// TwinCAT 3 PLC project ControlExtrusora
// ProgramVersion: 3.1.4023.0
// libraries:
//   Tc2_Standard, * (Beckhoff Automation GmbH)
//   Tc2_System, * (Beckhoff Automation GmbH)
//   Tc3_Module, * (Beckhoff Automation GmbH)
// project tree:
//   DUTs/ Modes.TcDUT (not stored)
//   / GlobalTextList.TcGTLO (not stored), PlcTask.TcTTO (not stored), Visualization Manager.TcVMO (not stored)
//   GVLs/ GVL.TcGVL (not stored), HMI.TcGVL (not stored), IO.TcGVL
//   POUs/ MAIN.TcPOU, OperatingModes.TcPOU
//   POUs/VISUCode/ VisuLogic.TcPOU (not stored)
//   VISUs/ MainHMI.TcVIS (not stored)
// real-time tasks:
//   TASK PlcTask: cycle T#10ms, priority 20, ADS port 350

// ---- GVLs/IO.TcGVL
{attribute 'qualified_only'}
VAR_GLOBAL
	
	// Termo-resistances outputs
	O_TermL:BOOL;
	O_TermU:BOOL;
END_VAR

// ---- POUs/MAIN.TcPOU
PROGRAM MAIN
VAR
	luz:BOOL:=TRUE;
END_VAR

Luz :=Luz;

END_PROGRAM

// ---- POUs/OperatingModes.TcPOU
PROGRAM OperatingModes
VAR
	aux:BOOL;
END_VAR

CASE GVL.Mode OF
	
	// Emergency stop
	Modes.STOP_EM:
		IF HMI.Bt_Rearm THEN
			gvl.Mode := modes.STOP_OP;
		END_IF
	
	// Operative stop
	Modes.STOP_OP:
		IF HMI.Bt_EmStop THEN
			GVL.Mode := Modes.STOP_EM;
		END_IF
		IF HMI.Bt_Run AND HMI.Sel_ManAuto THEN
			GVL.Mode := Modes.AUTO;
		END_IF
		IF NOT HMI.Sel_ManAuto THEN
			GVL.Mode := Modes.MAN;
		END_IF
		
	// Automatic
	Modes.AUTO:
		IF HMI.Bt_EmStop THEN
			GVL.Mode := Modes.STOP_EM;
		END_IF
		IF NOT HMI.Sel_ManAuto THEN
			GVL.Mode := Modes.MAN;
		END_IF
		IF HMI.Bt_Stop THEN
			GVL.Mode := Modes.STOP_OP;
		END_IF
		
	// Manual
	Modes.MAN:
		IF HMI.Bt_EmStop THEN
			GVL.Mode := Modes.STOP_EM;
		END_IF
		IF HMi.Sel_ManAuto THEN
			GVL.Mode := Modes.STOP_OP;
		END_IF
		
END_CASE

END_PROGRAM
